Universal Robots PolyScope program: wrs2020_taskboard_retainer_and_nut.urp

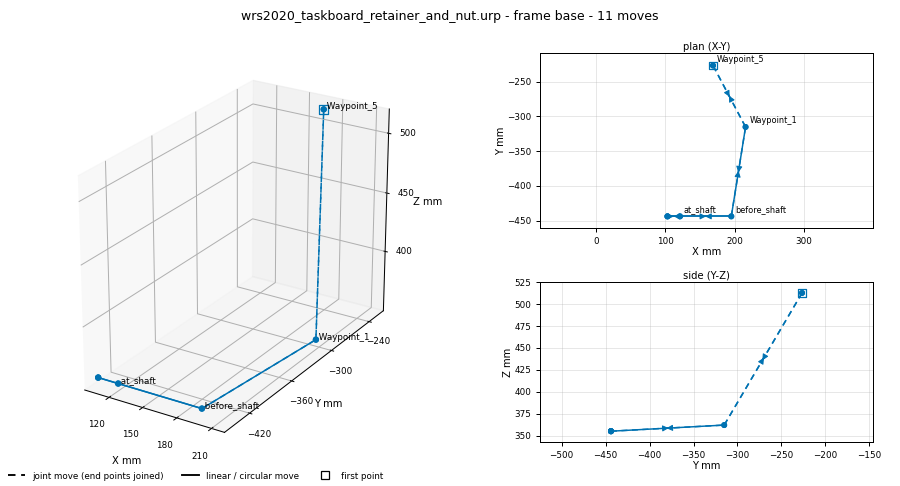
[picture p0: tool path of wrs2020_taskboard_retainer_and_nut.urp in frame base, 11 of 11 moves have a stored position in this frame; points joined in program order, loops and branches not executed]
Program wrs2020_taskboard_retainer_and_nut (installation=default directory=/programs createdIn=5.7.0.90932 lastSavedIn=5.7.0.90932 robotSerialNumber=20205500607)
Calibrated DH parameters: a=[0.000096, -0.337, -0.383372, 0.000118, 0.000015, 0]; d=[0.162724, 79.377998, -95.545185, 16.300583, 0.099689, 0.099499]; alpha=[1.569249, 0.003272, 0.005201, 1.570041, -1.570219, 0]; deltaTheta=[0, 0.65664, 5.410619, 0.215927, -0.000001, 0]
Robot Program (runOnlyOnce=true)
  MoveJ speed 120 deg/s, acceleration 150 deg/s^2 (useActiveTCP=false) tcp=TCP; feature=Base
    Waypoint Waypoint_5: TCP in base x=168.883 y=-226.544 z=512.618 mm, rx=-1.3574 ry=-2.6372 rz=0.1933 rad; joints [103.757, -121.415, 108.773, -76.619, -102.008, 68.039] deg
    Waypoint Waypoint_1: TCP in base x=215.797 y=-315.094 z=362.315 mm, rx=-2.0274 ry=-2.0144 rz=0.8026 rad; joints [112.634, -103.402, 123.505, -112.948, -122.464, 112.103] deg
  MoveL speed 250 mm/s, acceleration 1200 mm/s^2 (useActiveTCP=false) tcp=TCP; feature=Base
    Waypoint before_shaft: motionParameters(jointSpeed=1.047198 jointAcceleration=1.396263 cartesianSpeed=0.25 cartesianAcceleration=1.2); TCP in base x=195.25 y=-443.905 z=355.353 mm, rx=-2.2407 ry=-1.8942 rz=1.1081 rad; joints [105.164, -87.893, 117.051, -139.198, -126.623, 108.098] deg
    Waypoint at_shaft: motionParameters(jointSpeed=1.047198 jointAcceleration=1.396263 cartesianSpeed=0.035 cartesianAcceleration=1.2); TCP in base x=121.328 y=-443.905 z=355.353 mm, rx=-2.2407 ry=-1.8942 rz=1.1081 rad; joints [95.554, -91.325, 122.189, -147.104, -122.834, 97.339] deg
    Waypoint inside_shaft: motionParameters(jointSpeed=1.047198 jointAcceleration=1.396263 cartesianSpeed=0.005 cartesianAcceleration=1.2); TCP in base x=103.192 y=-443.905 z=355.353 mm, rx=-2.2407 ry=-1.8942 rz=1.1081 rad; joints [93.042, -91.968, 123.187, -148.887, -121.695, 94.691] deg
  Popup Message (haltProgram=false message=turn on motor, then press ok to fiddle bit into pulley inputType=Text)
  MoveL speed 1 mm/s, acceleration 10 mm/s^2 (useActiveTCP=false) tcp=TCP; feature=Base
    MoveDirectionNode (selectedDirection=YPlus)
      Until DISTANCE (allowActions=false deceleration=3 distanceNodeType=STOP) Distance=0.001; motionParameters(blendRadius=0)
    MoveDirectionNode (selectedDirection=YMinus)
      Until DISTANCE (allowActions=false deceleration=3 distanceNodeType=STOP) Distance=0.002; motionParameters(blendRadius=0)
    MoveDirectionNode (selectedDirection=YPlus toolParams=0.25, 1.2)
      Until DISTANCE (allowActions=false deceleration=3 distanceNodeType=STOP) Distance=0.001; motionParameters(blendRadius=0)
    MoveDirectionNode (selectedDirection=ZMinus)
      Until DISTANCE (allowActions=false deceleration=3 distanceNodeType=STOP) Distance=0.001; motionParameters(blendRadius=0)
    MoveDirectionNode (selectedDirection=ZPlus)
      Until DISTANCE (allowActions=false deceleration=3 distanceNodeType=STOP) Distance=0.002; motionParameters(blendRadius=0)
    MoveDirectionNode (selectedDirection=ZMinus)
      Until DISTANCE (allowActions=false deceleration=3 distanceNodeType=STOP) Distance=0.001; motionParameters(blendRadius=0)
    Waypoint inside_shaft: motionParameters(jointSpeed=1.047198 jointAcceleration=1.396263 cartesianSpeed=0.005 cartesianAcceleration=1.2); TCP in base x=103.192 y=-443.905 z=355.353 mm, rx=-2.2407 ry=-1.8942 rz=1.1081 rad; joints [93.042, -91.968, 123.187, -148.887, -121.695, 94.691] deg
  Popup Message (haltProgram=false message=wait until nut placed, then turn on motor. press ok to retreat inputType=Text)
  MoveL speed 250 mm/s, acceleration 1200 mm/s^2 (useActiveTCP=false) tcp=TCP; feature=Base
    Waypoint inside_shaft: motionParameters(jointSpeed=1.047198 jointAcceleration=1.396263 cartesianSpeed=0.005 cartesianAcceleration=1.2); TCP in base x=103.192 y=-443.905 z=355.353 mm, rx=-2.2407 ry=-1.8942 rz=1.1081 rad; joints [93.042, -91.968, 123.187, -148.887, -121.695, 94.691] deg
    Waypoint at_shaft: motionParameters(jointSpeed=1.047198 jointAcceleration=1.396263 cartesianSpeed=0.035 cartesianAcceleration=1.2); TCP in base x=121.328 y=-443.905 z=355.353 mm, rx=-2.2407 ry=-1.8942 rz=1.1081 rad; joints [95.554, -91.325, 122.189, -147.104, -122.834, 97.339] deg
    Waypoint before_shaft: motionParameters(jointSpeed=1.047198 jointAcceleration=1.396263 cartesianSpeed=0.25 cartesianAcceleration=1.2); TCP in base x=195.25 y=-443.905 z=355.353 mm, rx=-2.2407 ry=-1.8942 rz=1.1081 rad; joints [105.164, -87.893, 117.051, -139.198, -126.623, 108.098] deg
  MoveJ speed 120 deg/s, acceleration 150 deg/s^2 (useActiveTCP=false) tcp=TCP; feature=Base
    Waypoint Waypoint_1: TCP in base x=215.797 y=-315.094 z=362.315 mm, rx=-2.0274 ry=-2.0144 rz=0.8026 rad; joints [112.634, -103.402, 123.505, -112.948, -122.464, 112.103] deg
    Waypoint Waypoint_5: TCP in base x=168.883 y=-226.544 z=512.618 mm, rx=-1.3574 ry=-2.6372 rz=0.1933 rad; joints [103.757, -121.415, 108.773, -76.619, -102.008, 68.039] deg
